Staubli VAL3: decodeMsgBody.pgx

public program decodeMsgBody()
  local bool l_bFlag
begin
  l_bFlag = false

  switch rosGenericMsg.header.nMsgType
    case 11
      call decTrajPt(l_bFlag)
    break
    case 14
      call decTrajPtFull(l_bFlag)
    break
    default
    break
  endSwitch

  if (l_bFlag)
    // move on to state 4: push motion into buffer
    nDataInState = 4
  else
    // error whilst decoding msg body...
    if (rosGenericMsg.header.nCommType == 2)
      switch rosGenericMsg.header.nMsgType
        case 11
          rosTrajPtAck.header.nReplyCode = 2
        break
        case 14
          rosTrajPtFAck.header.nReplyCode = 2
        break
        default
        break
      endSwitch
      // jump to state 5: sendAck()
      nDataInState = 5
    else
      // reset state machine, since no ACK is required
      nDataInState = 1
    endIf
  endIf
end
